PROGRAM P_AxisControl
VAR
END_VAR

//Axis Control program based on youtube series Twincat 3 NC Videos MB05a until MB17b plus MB22 by @electricalautomation https://www.youtube.com/watch?v=BxRAOdTks9I&list=PL762SfoJC-e8NbAUQ-H7a_TOdqrlBPCw4&index=25

IF G_Inputs.bManualModeSelector THEN
	Manual_mode();
ELSIF G_Inputs.bAutoModeSelector THEN
	Auto_mode();
ELSE
	Stop_mode();
END_IF

METHOD Auto_mode : BOOL
VAR_INPUT
END_VAR
//AXIS 1 Main arm actuator

G_AXIS1.lrBC_PowerOverride := 100;

G_AXIS1.bBC_ResetExe := G_Inputs.bJoystickLeftEnable OR G_Inputs.bGreenButton OR G_AXIS1.bBC_MoveAbsDone;

//Power Enable
G_AXIS1.bBC_PowerEnCmd := G_Inputs.bAutoModeSelector;
G_AXIS1.bBC_PowerEnNegative := G_Inputs.bAutoModeSelector;
G_AXIS1.bBC_PowerEnPositive := G_Inputs.bAutoModeSelector;

G_AXIS1.lrBC_MoveAbsPosition := G_InverseKinematics.fStrokeActuatorMainInverse*1000;
G_AXIS1.lrBC_MoveAbsVelocity := 20;
G_AXIS1.bBC_MoveAbsExe := G_Inputs.bGreenButton;


//Position control
IF G_Inputs.bJoystickLeftEnable AND G_AXIS1.bBC_MoveAbsDone THEN
	G_AXIS1.bBC_ExtSetGenDisExe := FALSE;
	G_AXIS1.bBC_ExtSetGenEnaExe := TRUE;
ELSE
	G_AXIS1.bBC_ExtSetGenDisExe := TRUE;
	G_AXIS1.bBC_ExtSetGenEnaExe := FALSE;
END_IF


G_AXIS1.lrBC_MoveAddPos := G_InverseKinematics.fStrokeActuatorMainInverse*1000;


//Update axis
AXIS1_LD_Auto();


//Axis 3 Knuckle arm actuator

G_AXIS3.lrTC_PowerOverride := 100;

G_AXIS3.bTC_ResetExe := G_Inputs.bJoystickLeftEnable OR G_Inputs.bGreenButton OR G_AXIS3.bTC_MoveAbsDone;

//Power Enable
G_AXIS3.bTC_PowerEnCmd := G_Inputs.bAutoModeSelector;
G_AXIS3.bTC_PowerEnNegative := G_Inputs.bAutoModeSelector;
G_AXIS3.bTC_PowerEnPositive := G_Inputs.bAutoModeSelector;

G_AXIS3.lrTC_MoveAbsPosition := G_InverseKinematics.fStrokeActuatorKnuckleInverse*1000;
G_AXIS3.lrTC_MoveAbsVelocity := 20;
G_AXIS3.bTC_MoveAbsExe := G_Inputs.bGreenButton;


//Position control
IF G_Inputs.bJoystickLeftEnable AND G_AXIS3.bTC_MoveAbsDone THEN
	G_AXIS3.bTC_ExtSetGenDisExe := FALSE;
	G_AXIS3.bTC_ExtSetGenEnaExe := TRUE;
ELSE
	G_AXIS3.bTC_ExtSetGenDisExe := TRUE;
	G_AXIS3.bTC_ExtSetGenEnaExe := FALSE;
END_IF


G_AXIS3.lrTC_MoveAddPos := G_InverseKinematics.fStrokeActuatorKnuckleInverse*1000;


//Update axis
AXIS3_LD_Auto();


//Axis 4 Winch motor

G_AXIS4.lrWM_PowerOverride := 50;

G_AXIS4.bWM_ResetExe := G_Inputs.bGreenButton OR G_AXIS1.bBC_MoveAbsDone;
//GVL_AXIS4.bWM_ResetExe := G_Inputs.bJoystickRightEnable OR G_Inputs.bGreenButton OR GVL_AXIS1.bBC_MoveAbsDone;

//Power Enable
G_AXIS4.bWM_PowerEnCmd := G_Inputs.bAutoModeSelector;
G_AXIS4.bWM_PowerEnNegative := G_Inputs.bAutoModeSelector;
G_AXIS4.bWM_PowerEnPositive := G_Inputs.bAutoModeSelector;

//G_AXIS4.lrWM_MoveAbsPosition := G_MachineControl.fWinchMotorAngleRef*180/PI;
//G_AXIS4.lrWM_MoveAbsVelocity := 50;
//G_AXIS4.bWM_MoveAbsExe := G_Inputs.bGreenButton;

//Position control
IF G_Inputs.bJoystickLeftEnable AND G_AXIS1.bBC_MoveAbsDone AND G_AXIS3.bTC_MoveAbsDone THEN
	G_AXIS4.bWM_ExtSetGenDisExe := FALSE;
	G_AXIS4.bWM_ExtSetGenEnaExe := TRUE;
ELSE
	G_AXIS4.bWM_ExtSetGenDisExe := TRUE;
	G_AXIS4.bWM_ExtSetGenEnaExe := FALSE;
END_IF

G_AXIS4.lrWM_MoveSetPointVel := 500;
G_AXIS4.lrWM_MoveAddPos := G_MachineControl.fWinchMotorAngleAbsRef; //G_MachineControl.fWinchMotorAngleRef*180/PI; //Convert to degrees


//Update axis
AXIS4_LD_Auto();
END_METHOD

METHOD AXIS1_LD_Auto : BOOL
VAR_INPUT
END_VAR
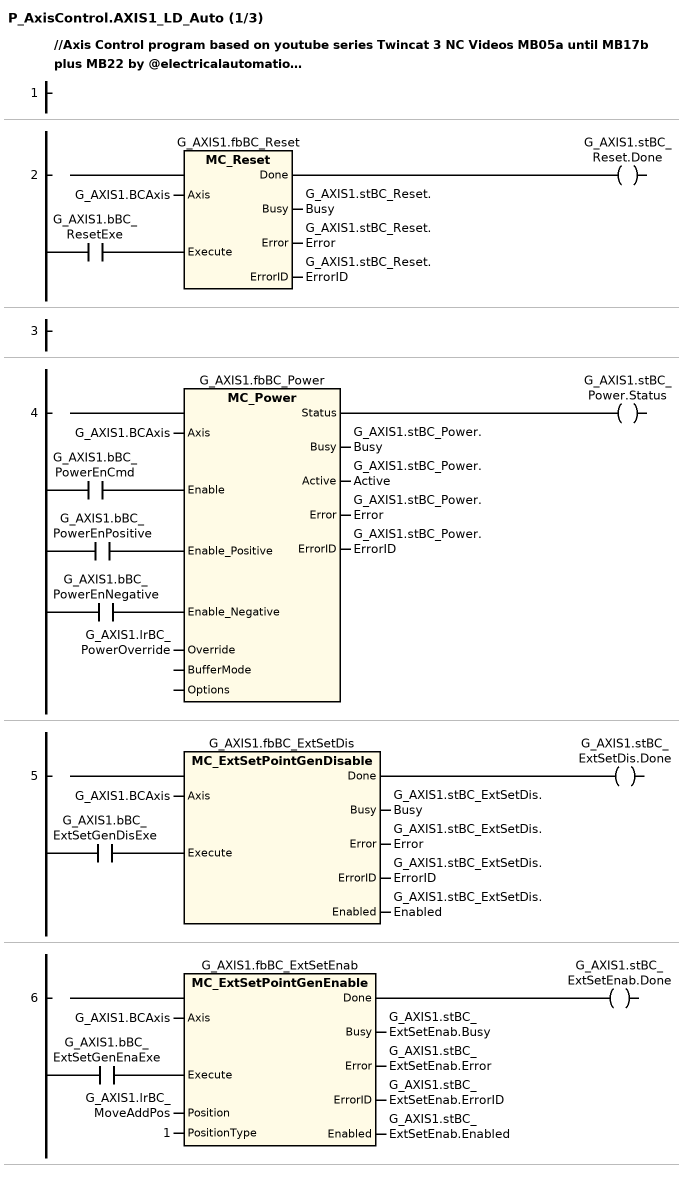
// NETWORK 1: //Axis Control program based on youtube series Twincat 3 NC Videos MB05a until MB17b plus MB22 by @electricalautomation https://www.youtube.com/watch?v=BxRAOdTks9I&list=PL762SfoJC-e8NbAUQ-H7a_TOdqrlBPCw4&index=25

// NETWORK 2
G_AXIS1.fbBC_Reset(
    Axis := G_AXIS1.BCAxis,
    Execute := G_AXIS1.bBC_ResetExe,
    Busy => G_AXIS1.stBC_Reset.Busy,
    Error => G_AXIS1.stBC_Reset.Error,
    ErrorID => G_AXIS1.stBC_Reset.ErrorID); // MC_Reset
G_AXIS1.stBC_Reset.Done := G_AXIS1.fbBC_Reset.Done;

// NETWORK 3

// NETWORK 4
G_AXIS1.fbBC_Power(
    Axis := G_AXIS1.BCAxis,
    Enable := G_AXIS1.bBC_PowerEnCmd,
    Enable_Positive := G_AXIS1.bBC_PowerEnPositive,
    Enable_Negative := G_AXIS1.bBC_PowerEnNegative,
    Override := G_AXIS1.lrBC_PowerOverride,
    Busy => G_AXIS1.stBC_Power.Busy,
    Active => G_AXIS1.stBC_Power.Active,
    Error => G_AXIS1.stBC_Power.Error,
    ErrorID => G_AXIS1.stBC_Power.ErrorID); // MC_Power
G_AXIS1.stBC_Power.Status := G_AXIS1.fbBC_Power.Status;

// NETWORK 5
G_AXIS1.fbBC_ExtSetDis(
    Axis := G_AXIS1.BCAxis,
    Execute := G_AXIS1.bBC_ExtSetGenDisExe,
    Busy => G_AXIS1.stBC_ExtSetDis.Busy,
    Error => G_AXIS1.stBC_ExtSetDis.Error,
    ErrorID => G_AXIS1.stBC_ExtSetDis.ErrorID,
    Enabled => G_AXIS1.stBC_ExtSetDis.Enabled); // MC_ExtSetPointGenDisable
G_AXIS1.stBC_ExtSetDis.Done := G_AXIS1.fbBC_ExtSetDis.Done;

// NETWORK 6
G_AXIS1.fbBC_ExtSetEnab(
    Axis := G_AXIS1.BCAxis,
    Execute := G_AXIS1.bBC_ExtSetGenEnaExe,
    Position := G_AXIS1.lrBC_MoveAddPos,
    PositionType := 1,
    Busy => G_AXIS1.stBC_ExtSetEnab.Busy,
    Error => G_AXIS1.stBC_ExtSetEnab.Error,
    ErrorID => G_AXIS1.stBC_ExtSetEnab.ErrorID,
    Enabled => G_AXIS1.stBC_ExtSetEnab.Enabled); // MC_ExtSetPointGenEnable
G_AXIS1.stBC_ExtSetEnab.Done := G_AXIS1.fbBC_ExtSetEnab.Done;

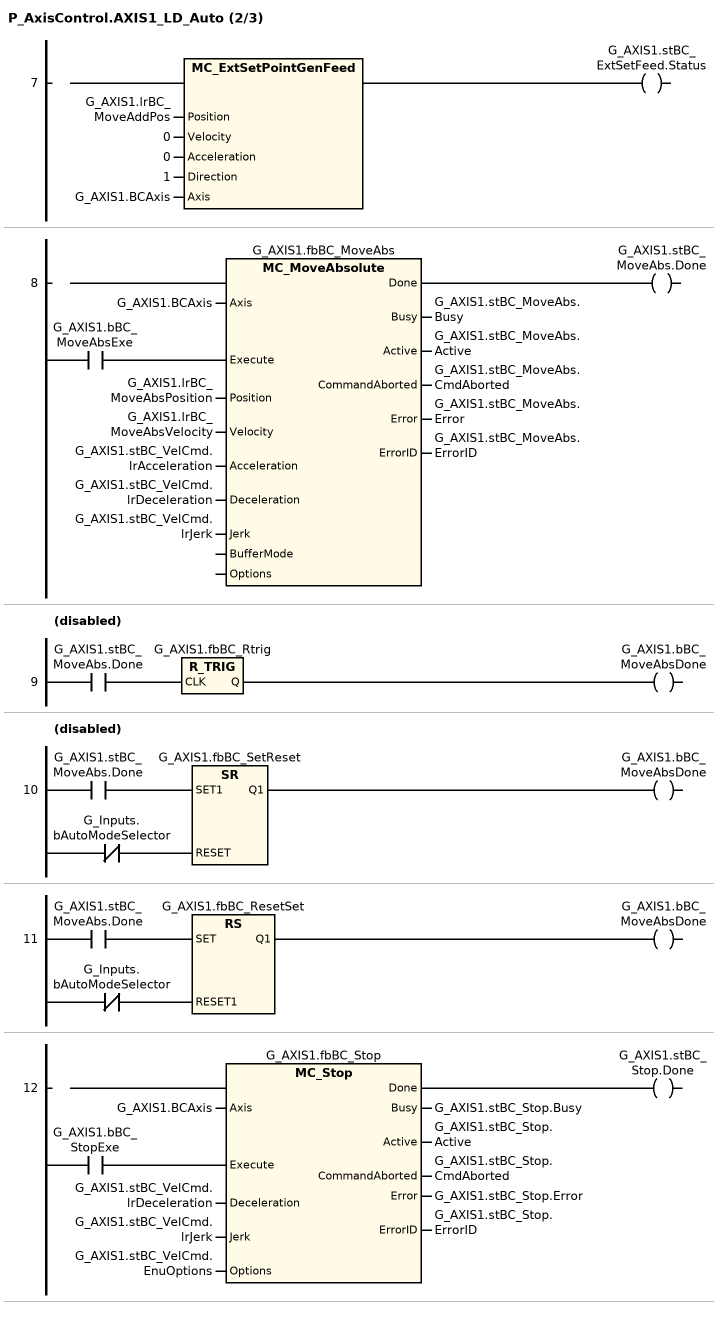
// NETWORK 7
G_AXIS1.stBC_ExtSetFeed.Status := MC_ExtSetPointGenFeed(Position := G_AXIS1.lrBC_MoveAddPos, Velocity := 0, Acceleration := 0, Direction := 1, Axis := G_AXIS1.BCAxis);

// NETWORK 8
G_AXIS1.fbBC_MoveAbs(
    Axis := G_AXIS1.BCAxis,
    Execute := G_AXIS1.bBC_MoveAbsExe,
    Position := G_AXIS1.lrBC_MoveAbsPosition,
    Velocity := G_AXIS1.lrBC_MoveAbsVelocity,
    Acceleration := G_AXIS1.stBC_VelCmd.lrAcceleration,
    Deceleration := G_AXIS1.stBC_VelCmd.lrDeceleration,
    Jerk := G_AXIS1.stBC_VelCmd.lrJerk,
    Busy => G_AXIS1.stBC_MoveAbs.Busy,
    Active => G_AXIS1.stBC_MoveAbs.Active,
    CommandAborted => G_AXIS1.stBC_MoveAbs.CmdAborted,
    Error => G_AXIS1.stBC_MoveAbs.Error,
    ErrorID => G_AXIS1.stBC_MoveAbs.ErrorID); // MC_MoveAbsolute
G_AXIS1.stBC_MoveAbs.Done := G_AXIS1.fbBC_MoveAbs.Done;

// NETWORK 9 (disabled)
// G_AXIS1.fbBC_Rtrig(CLK := G_AXIS1.stBC_MoveAbs.Done); // R_TRIG
// G_AXIS1.bBC_MoveAbsDone := G_AXIS1.fbBC_Rtrig.Q;

// NETWORK 10 (disabled)
// G_AXIS1.fbBC_SetReset(SET1 := G_AXIS1.stBC_MoveAbs.Done, RESET := NOT G_Inputs.bAutoModeSelector); // SR
// G_AXIS1.bBC_MoveAbsDone := G_AXIS1.fbBC_SetReset.Q1;

// NETWORK 11
G_AXIS1.fbBC_ResetSet(SET := G_AXIS1.stBC_MoveAbs.Done, RESET1 := NOT G_Inputs.bAutoModeSelector); // RS
G_AXIS1.bBC_MoveAbsDone := G_AXIS1.fbBC_ResetSet.Q1;

// NETWORK 12
G_AXIS1.fbBC_Stop(
    Axis := G_AXIS1.BCAxis,
    Execute := G_AXIS1.bBC_StopExe,
    Deceleration := G_AXIS1.stBC_VelCmd.lrDeceleration,
    Jerk := G_AXIS1.stBC_VelCmd.lrJerk,
    Options := G_AXIS1.stBC_VelCmd.EnuOptions,
    Busy => G_AXIS1.stBC_Stop.Busy,
    Active => G_AXIS1.stBC_Stop.Active,
    CommandAborted => G_AXIS1.stBC_Stop.CmdAborted,
    Error => G_AXIS1.stBC_Stop.Error,
    ErrorID => G_AXIS1.stBC_Stop.ErrorID); // MC_Stop
G_AXIS1.stBC_Stop.Done := G_AXIS1.fbBC_Stop.Done;

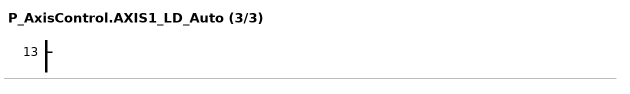
// NETWORK 13
END_METHOD

METHOD AXIS1_LD_Manual : BOOL
VAR_INPUT
END_VAR
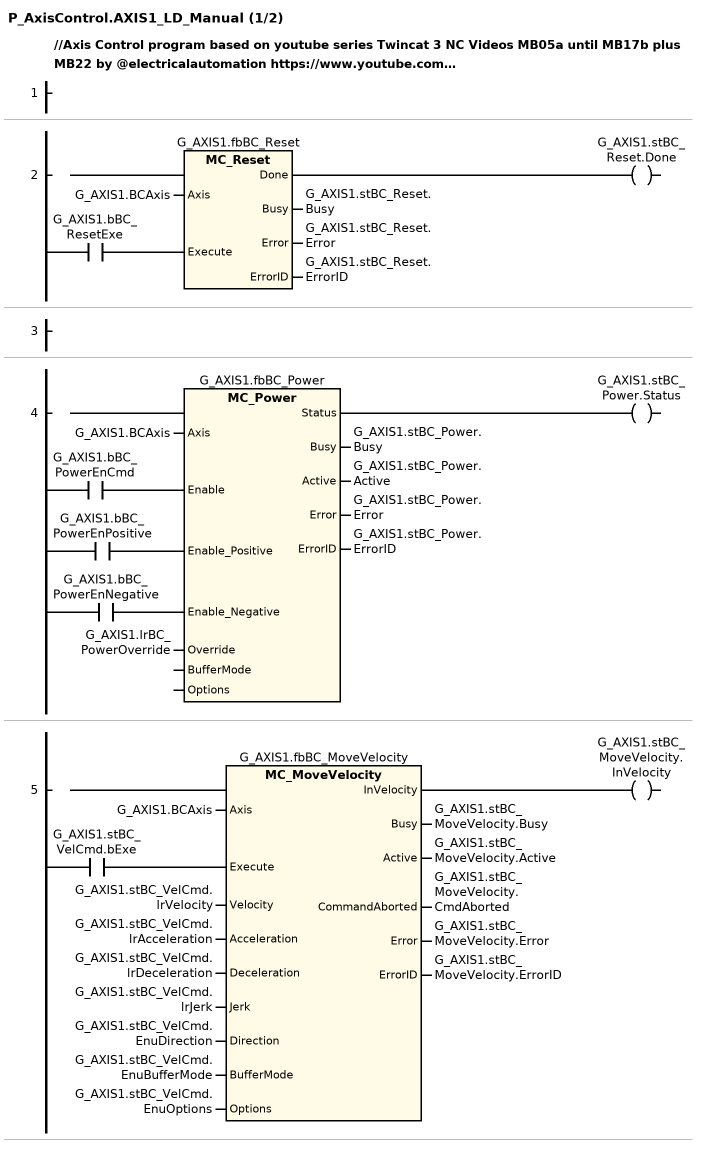
// NETWORK 1: //Axis Control program based on youtube series Twincat 3 NC Videos MB05a until MB17b plus MB22 by @electricalautomation https://www.youtube.com/watch?v=BxRAOdTks9I&list=PL762SfoJC-e8NbAUQ-H7a_TOdqrlBPCw4&index=25

// NETWORK 2
G_AXIS1.fbBC_Reset(
    Axis := G_AXIS1.BCAxis,
    Execute := G_AXIS1.bBC_ResetExe,
    Busy => G_AXIS1.stBC_Reset.Busy,
    Error => G_AXIS1.stBC_Reset.Error,
    ErrorID => G_AXIS1.stBC_Reset.ErrorID); // MC_Reset
G_AXIS1.stBC_Reset.Done := G_AXIS1.fbBC_Reset.Done;

// NETWORK 3

// NETWORK 4
G_AXIS1.fbBC_Power(
    Axis := G_AXIS1.BCAxis,
    Enable := G_AXIS1.bBC_PowerEnCmd,
    Enable_Positive := G_AXIS1.bBC_PowerEnPositive,
    Enable_Negative := G_AXIS1.bBC_PowerEnNegative,
    Override := G_AXIS1.lrBC_PowerOverride,
    Busy => G_AXIS1.stBC_Power.Busy,
    Active => G_AXIS1.stBC_Power.Active,
    Error => G_AXIS1.stBC_Power.Error,
    ErrorID => G_AXIS1.stBC_Power.ErrorID); // MC_Power
G_AXIS1.stBC_Power.Status := G_AXIS1.fbBC_Power.Status;

// NETWORK 5
G_AXIS1.fbBC_MoveVelocity(
    Axis := G_AXIS1.BCAxis,
    Execute := G_AXIS1.stBC_VelCmd.bExe,
    Velocity := G_AXIS1.stBC_VelCmd.lrVelocity,
    Acceleration := G_AXIS1.stBC_VelCmd.lrAcceleration,
    Deceleration := G_AXIS1.stBC_VelCmd.lrDeceleration,
    Jerk := G_AXIS1.stBC_VelCmd.lrJerk,
    Direction := G_AXIS1.stBC_VelCmd.EnuDirection,
    BufferMode := G_AXIS1.stBC_VelCmd.EnuBufferMode,
    Options := G_AXIS1.stBC_VelCmd.EnuOptions,
    Busy => G_AXIS1.stBC_MoveVelocity.Busy,
    Active => G_AXIS1.stBC_MoveVelocity.Active,
    CommandAborted => G_AXIS1.stBC_MoveVelocity.CmdAborted,
    Error => G_AXIS1.stBC_MoveVelocity.Error,
    ErrorID => G_AXIS1.stBC_MoveVelocity.ErrorID); // MC_MoveVelocity
G_AXIS1.stBC_MoveVelocity.InVelocity := G_AXIS1.fbBC_MoveVelocity.InVelocity;

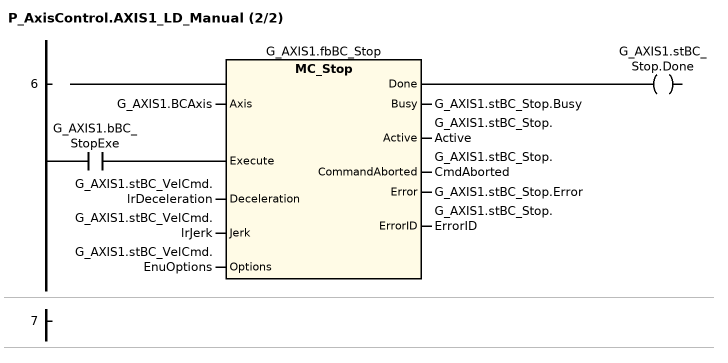
// NETWORK 6
G_AXIS1.fbBC_Stop(
    Axis := G_AXIS1.BCAxis,
    Execute := G_AXIS1.bBC_StopExe,
    Deceleration := G_AXIS1.stBC_VelCmd.lrDeceleration,
    Jerk := G_AXIS1.stBC_VelCmd.lrJerk,
    Options := G_AXIS1.stBC_VelCmd.EnuOptions,
    Busy => G_AXIS1.stBC_Stop.Busy,
    Active => G_AXIS1.stBC_Stop.Active,
    CommandAborted => G_AXIS1.stBC_Stop.CmdAborted,
    Error => G_AXIS1.stBC_Stop.Error,
    ErrorID => G_AXIS1.stBC_Stop.ErrorID); // MC_Stop
G_AXIS1.stBC_Stop.Done := G_AXIS1.fbBC_Stop.Done;

// NETWORK 7
END_METHOD

METHOD AXIS2_LD_Manual : BOOL
VAR_INPUT
END_VAR
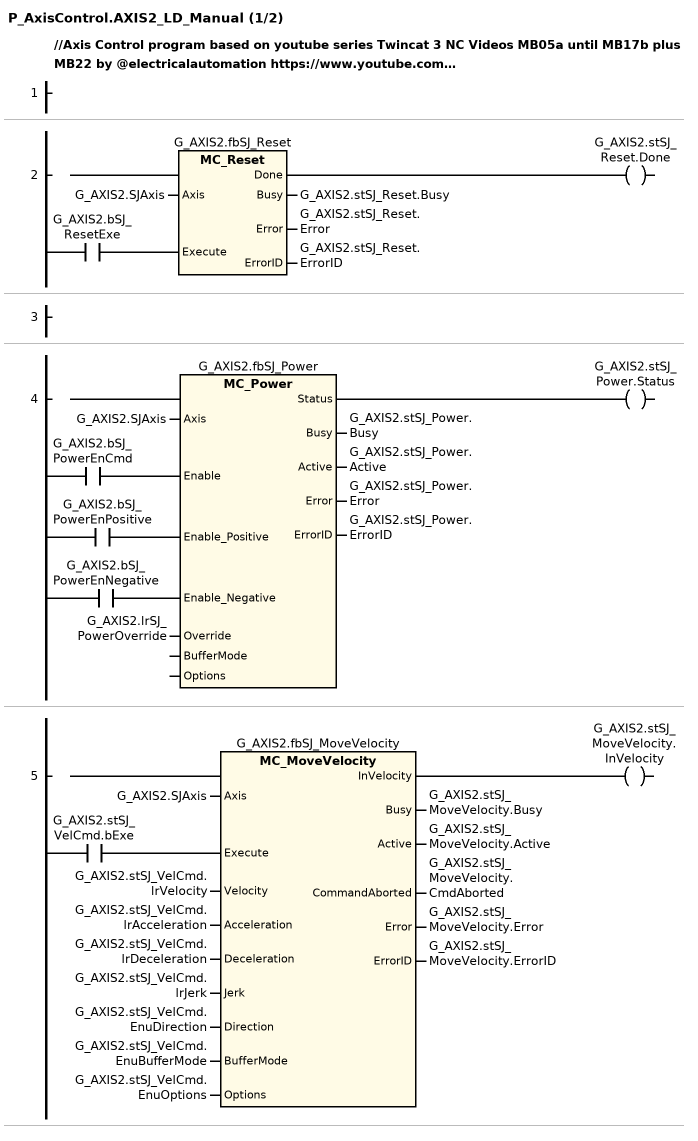
// NETWORK 1: //Axis Control program based on youtube series Twincat 3 NC Videos MB05a until MB17b plus MB22 by @electricalautomation https://www.youtube.com/watch?v=BxRAOdTks9I&list=PL762SfoJC-e8NbAUQ-H7a_TOdqrlBPCw4&index=25

// NETWORK 2
G_AXIS2.fbSJ_Reset(
    Axis := G_AXIS2.SJAxis,
    Execute := G_AXIS2.bSJ_ResetExe,
    Busy => G_AXIS2.stSJ_Reset.Busy,
    Error => G_AXIS2.stSJ_Reset.Error,
    ErrorID => G_AXIS2.stSJ_Reset.ErrorID); // MC_Reset
G_AXIS2.stSJ_Reset.Done := G_AXIS2.fbSJ_Reset.Done;

// NETWORK 3

// NETWORK 4
G_AXIS2.fbSJ_Power(
    Axis := G_AXIS2.SJAxis,
    Enable := G_AXIS2.bSJ_PowerEnCmd,
    Enable_Positive := G_AXIS2.bSJ_PowerEnPositive,
    Enable_Negative := G_AXIS2.bSJ_PowerEnNegative,
    Override := G_AXIS2.lrSJ_PowerOverride,
    Busy => G_AXIS2.stSJ_Power.Busy,
    Active => G_AXIS2.stSJ_Power.Active,
    Error => G_AXIS2.stSJ_Power.Error,
    ErrorID => G_AXIS2.stSJ_Power.ErrorID); // MC_Power
G_AXIS2.stSJ_Power.Status := G_AXIS2.fbSJ_Power.Status;

// NETWORK 5
G_AXIS2.fbSJ_MoveVelocity(
    Axis := G_AXIS2.SJAxis,
    Execute := G_AXIS2.stSJ_VelCmd.bExe,
    Velocity := G_AXIS2.stSJ_VelCmd.lrVelocity,
    Acceleration := G_AXIS2.stSJ_VelCmd.lrAcceleration,
    Deceleration := G_AXIS2.stSJ_VelCmd.lrDeceleration,
    Jerk := G_AXIS2.stSJ_VelCmd.lrJerk,
    Direction := G_AXIS2.stSJ_VelCmd.EnuDirection,
    BufferMode := G_AXIS2.stSJ_VelCmd.EnuBufferMode,
    Options := G_AXIS2.stSJ_VelCmd.EnuOptions,
    Busy => G_AXIS2.stSJ_MoveVelocity.Busy,
    Active => G_AXIS2.stSJ_MoveVelocity.Active,
    CommandAborted => G_AXIS2.stSJ_MoveVelocity.CmdAborted,
    Error => G_AXIS2.stSJ_MoveVelocity.Error,
    ErrorID => G_AXIS2.stSJ_MoveVelocity.ErrorID); // MC_MoveVelocity
G_AXIS2.stSJ_MoveVelocity.InVelocity := G_AXIS2.fbSJ_MoveVelocity.InVelocity;

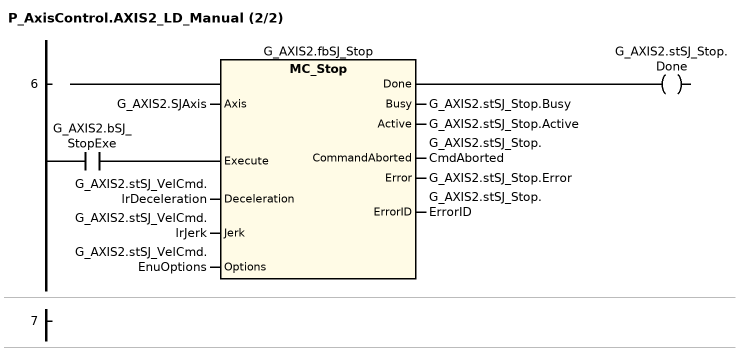
// NETWORK 6
G_AXIS2.fbSJ_Stop(
    Axis := G_AXIS2.SJAxis,
    Execute := G_AXIS2.bSJ_StopExe,
    Deceleration := G_AXIS2.stSJ_VelCmd.lrDeceleration,
    Jerk := G_AXIS2.stSJ_VelCmd.lrJerk,
    Options := G_AXIS2.stSJ_VelCmd.EnuOptions,
    Busy => G_AXIS2.stSJ_Stop.Busy,
    Active => G_AXIS2.stSJ_Stop.Active,
    CommandAborted => G_AXIS2.stSJ_Stop.CmdAborted,
    Error => G_AXIS2.stSJ_Stop.Error,
    ErrorID => G_AXIS2.stSJ_Stop.ErrorID); // MC_Stop
G_AXIS2.stSJ_Stop.Done := G_AXIS2.fbSJ_Stop.Done;

// NETWORK 7
END_METHOD

METHOD AXIS3_LD_Auto : BOOL
VAR_INPUT
END_VAR
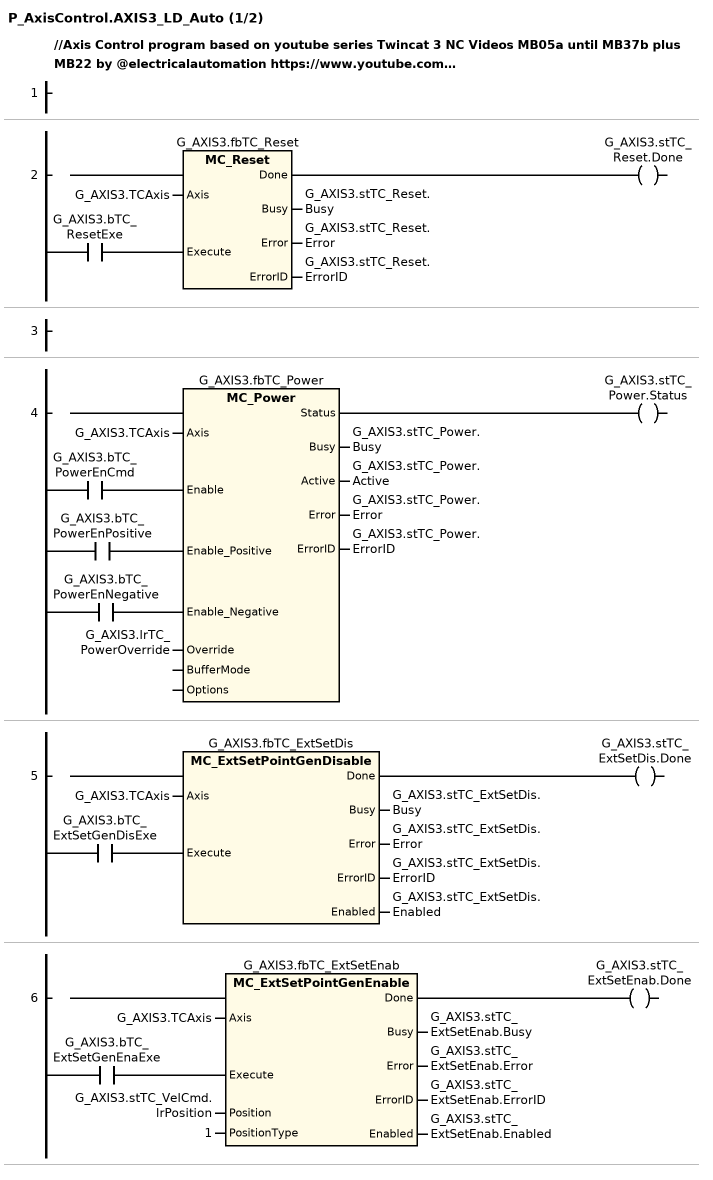
// NETWORK 1: //Axis Control program based on youtube series Twincat 3 NC Videos MB05a until MB37b plus MB22 by @electricalautomation https://www.youtube.com/watch?v=BxRAOdTks9I&list=PL762SfoJC-e8NbAUQ-H7a_TOdqrlBPCw4&index=25

// NETWORK 2
G_AXIS3.fbTC_Reset(
    Axis := G_AXIS3.TCAxis,
    Execute := G_AXIS3.bTC_ResetExe,
    Busy => G_AXIS3.stTC_Reset.Busy,
    Error => G_AXIS3.stTC_Reset.Error,
    ErrorID => G_AXIS3.stTC_Reset.ErrorID); // MC_Reset
G_AXIS3.stTC_Reset.Done := G_AXIS3.fbTC_Reset.Done;

// NETWORK 3

// NETWORK 4
G_AXIS3.fbTC_Power(
    Axis := G_AXIS3.TCAxis,
    Enable := G_AXIS3.bTC_PowerEnCmd,
    Enable_Positive := G_AXIS3.bTC_PowerEnPositive,
    Enable_Negative := G_AXIS3.bTC_PowerEnNegative,
    Override := G_AXIS3.lrTC_PowerOverride,
    Busy => G_AXIS3.stTC_Power.Busy,
    Active => G_AXIS3.stTC_Power.Active,
    Error => G_AXIS3.stTC_Power.Error,
    ErrorID => G_AXIS3.stTC_Power.ErrorID); // MC_Power
G_AXIS3.stTC_Power.Status := G_AXIS3.fbTC_Power.Status;

// NETWORK 5
G_AXIS3.fbTC_ExtSetDis(
    Axis := G_AXIS3.TCAxis,
    Execute := G_AXIS3.bTC_ExtSetGenDisExe,
    Busy => G_AXIS3.stTC_ExtSetDis.Busy,
    Error => G_AXIS3.stTC_ExtSetDis.Error,
    ErrorID => G_AXIS3.stTC_ExtSetDis.ErrorID,
    Enabled => G_AXIS3.stTC_ExtSetDis.Enabled); // MC_ExtSetPointGenDisable
G_AXIS3.stTC_ExtSetDis.Done := G_AXIS3.fbTC_ExtSetDis.Done;

// NETWORK 6
G_AXIS3.fbTC_ExtSetEnab(
    Axis := G_AXIS3.TCAxis,
    Execute := G_AXIS3.bTC_ExtSetGenEnaExe,
    Position := G_AXIS3.stTC_VelCmd.lrPosition,
    PositionType := 1,
    Busy => G_AXIS3.stTC_ExtSetEnab.Busy,
    Error => G_AXIS3.stTC_ExtSetEnab.Error,
    ErrorID => G_AXIS3.stTC_ExtSetEnab.ErrorID,
    Enabled => G_AXIS3.stTC_ExtSetEnab.Enabled); // MC_ExtSetPointGenEnable
G_AXIS3.stTC_ExtSetEnab.Done := G_AXIS3.fbTC_ExtSetEnab.Done;

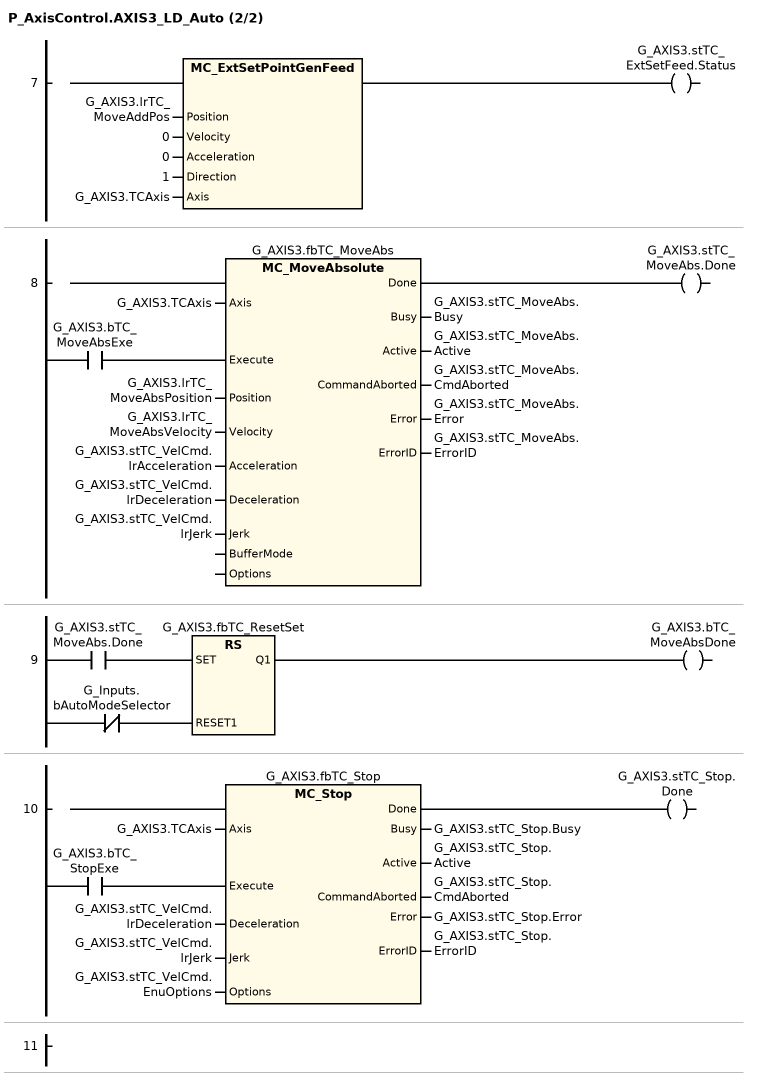
// NETWORK 7
G_AXIS3.stTC_ExtSetFeed.Status := MC_ExtSetPointGenFeed(Position := G_AXIS3.lrTC_MoveAddPos, Velocity := 0, Acceleration := 0, Direction := 1, Axis := G_AXIS3.TCAxis);

// NETWORK 8
G_AXIS3.fbTC_MoveAbs(
    Axis := G_AXIS3.TCAxis,
    Execute := G_AXIS3.bTC_MoveAbsExe,
    Position := G_AXIS3.lrTC_MoveAbsPosition,
    Velocity := G_AXIS3.lrTC_MoveAbsVelocity,
    Acceleration := G_AXIS3.stTC_VelCmd.lrAcceleration,
    Deceleration := G_AXIS3.stTC_VelCmd.lrDeceleration,
    Jerk := G_AXIS3.stTC_VelCmd.lrJerk,
    Busy => G_AXIS3.stTC_MoveAbs.Busy,
    Active => G_AXIS3.stTC_MoveAbs.Active,
    CommandAborted => G_AXIS3.stTC_MoveAbs.CmdAborted,
    Error => G_AXIS3.stTC_MoveAbs.Error,
    ErrorID => G_AXIS3.stTC_MoveAbs.ErrorID); // MC_MoveAbsolute
G_AXIS3.stTC_MoveAbs.Done := G_AXIS3.fbTC_MoveAbs.Done;

// NETWORK 9
G_AXIS3.fbTC_ResetSet(SET := G_AXIS3.stTC_MoveAbs.Done, RESET1 := NOT G_Inputs.bAutoModeSelector); // RS
G_AXIS3.bTC_MoveAbsDone := G_AXIS3.fbTC_ResetSet.Q1;

// NETWORK 10
G_AXIS3.fbTC_Stop(
    Axis := G_AXIS3.TCAxis,
    Execute := G_AXIS3.bTC_StopExe,
    Deceleration := G_AXIS3.stTC_VelCmd.lrDeceleration,
    Jerk := G_AXIS3.stTC_VelCmd.lrJerk,
    Options := G_AXIS3.stTC_VelCmd.EnuOptions,
    Busy => G_AXIS3.stTC_Stop.Busy,
    Active => G_AXIS3.stTC_Stop.Active,
    CommandAborted => G_AXIS3.stTC_Stop.CmdAborted,
    Error => G_AXIS3.stTC_Stop.Error,
    ErrorID => G_AXIS3.stTC_Stop.ErrorID); // MC_Stop
G_AXIS3.stTC_Stop.Done := G_AXIS3.fbTC_Stop.Done;

// NETWORK 11
END_METHOD

METHOD AXIS3_LD_Manual : BOOL
VAR_INPUT
END_VAR
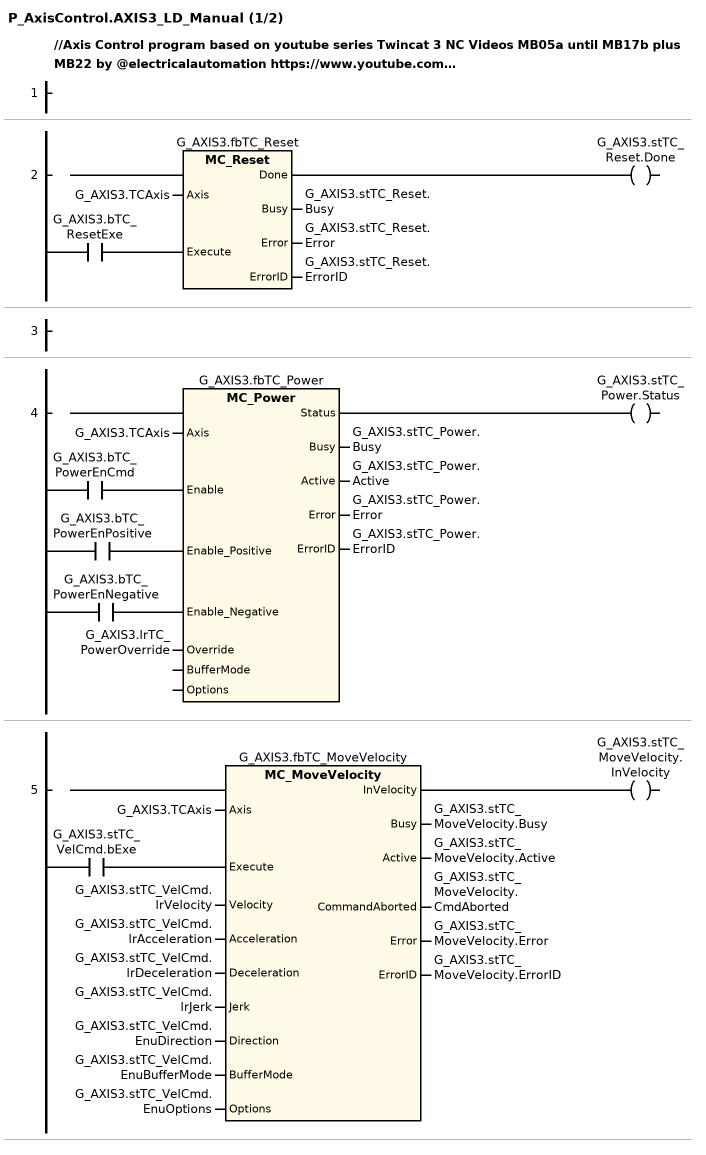
// NETWORK 1: //Axis Control program based on youtube series Twincat 3 NC Videos MB05a until MB17b plus MB22 by @electricalautomation https://www.youtube.com/watch?v=BxRAOdTks9I&list=PL762SfoJC-e8NbAUQ-H7a_TOdqrlBPCw4&index=25

// NETWORK 2
G_AXIS3.fbTC_Reset(
    Axis := G_AXIS3.TCAxis,
    Execute := G_AXIS3.bTC_ResetExe,
    Busy => G_AXIS3.stTC_Reset.Busy,
    Error => G_AXIS3.stTC_Reset.Error,
    ErrorID => G_AXIS3.stTC_Reset.ErrorID); // MC_Reset
G_AXIS3.stTC_Reset.Done := G_AXIS3.fbTC_Reset.Done;

// NETWORK 3

// NETWORK 4
G_AXIS3.fbTC_Power(
    Axis := G_AXIS3.TCAxis,
    Enable := G_AXIS3.bTC_PowerEnCmd,
    Enable_Positive := G_AXIS3.bTC_PowerEnPositive,
    Enable_Negative := G_AXIS3.bTC_PowerEnNegative,
    Override := G_AXIS3.lrTC_PowerOverride,
    Busy => G_AXIS3.stTC_Power.Busy,
    Active => G_AXIS3.stTC_Power.Active,
    Error => G_AXIS3.stTC_Power.Error,
    ErrorID => G_AXIS3.stTC_Power.ErrorID); // MC_Power
G_AXIS3.stTC_Power.Status := G_AXIS3.fbTC_Power.Status;

// NETWORK 5
G_AXIS3.fbTC_MoveVelocity(
    Axis := G_AXIS3.TCAxis,
    Execute := G_AXIS3.stTC_VelCmd.bExe,
    Velocity := G_AXIS3.stTC_VelCmd.lrVelocity,
    Acceleration := G_AXIS3.stTC_VelCmd.lrAcceleration,
    Deceleration := G_AXIS3.stTC_VelCmd.lrDeceleration,
    Jerk := G_AXIS3.stTC_VelCmd.lrJerk,
    Direction := G_AXIS3.stTC_VelCmd.EnuDirection,
    BufferMode := G_AXIS3.stTC_VelCmd.EnuBufferMode,
    Options := G_AXIS3.stTC_VelCmd.EnuOptions,
    Busy => G_AXIS3.stTC_MoveVelocity.Busy,
    Active => G_AXIS3.stTC_MoveVelocity.Active,
    CommandAborted => G_AXIS3.stTC_MoveVelocity.CmdAborted,
    Error => G_AXIS3.stTC_MoveVelocity.Error,
    ErrorID => G_AXIS3.stTC_MoveVelocity.ErrorID); // MC_MoveVelocity
G_AXIS3.stTC_MoveVelocity.InVelocity := G_AXIS3.fbTC_MoveVelocity.InVelocity;

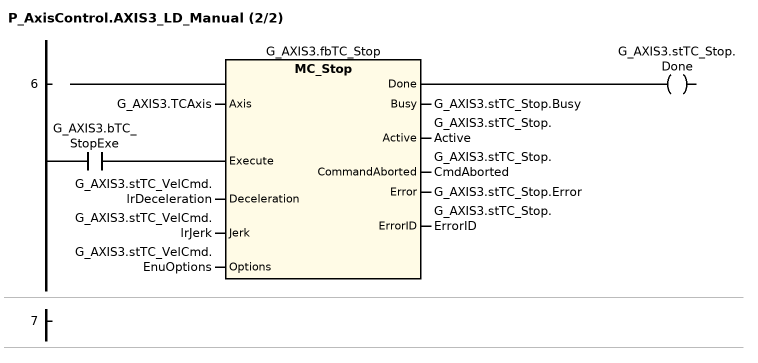
// NETWORK 6
G_AXIS3.fbTC_Stop(
    Axis := G_AXIS3.TCAxis,
    Execute := G_AXIS3.bTC_StopExe,
    Deceleration := G_AXIS3.stTC_VelCmd.lrDeceleration,
    Jerk := G_AXIS3.stTC_VelCmd.lrJerk,
    Options := G_AXIS3.stTC_VelCmd.EnuOptions,
    Busy => G_AXIS3.stTC_Stop.Busy,
    Active => G_AXIS3.stTC_Stop.Active,
    CommandAborted => G_AXIS3.stTC_Stop.CmdAborted,
    Error => G_AXIS3.stTC_Stop.Error,
    ErrorID => G_AXIS3.stTC_Stop.ErrorID); // MC_Stop
G_AXIS3.stTC_Stop.Done := G_AXIS3.fbTC_Stop.Done;

// NETWORK 7
END_METHOD

METHOD AXIS4_LD_Auto : BOOL
VAR_INPUT
END_VAR
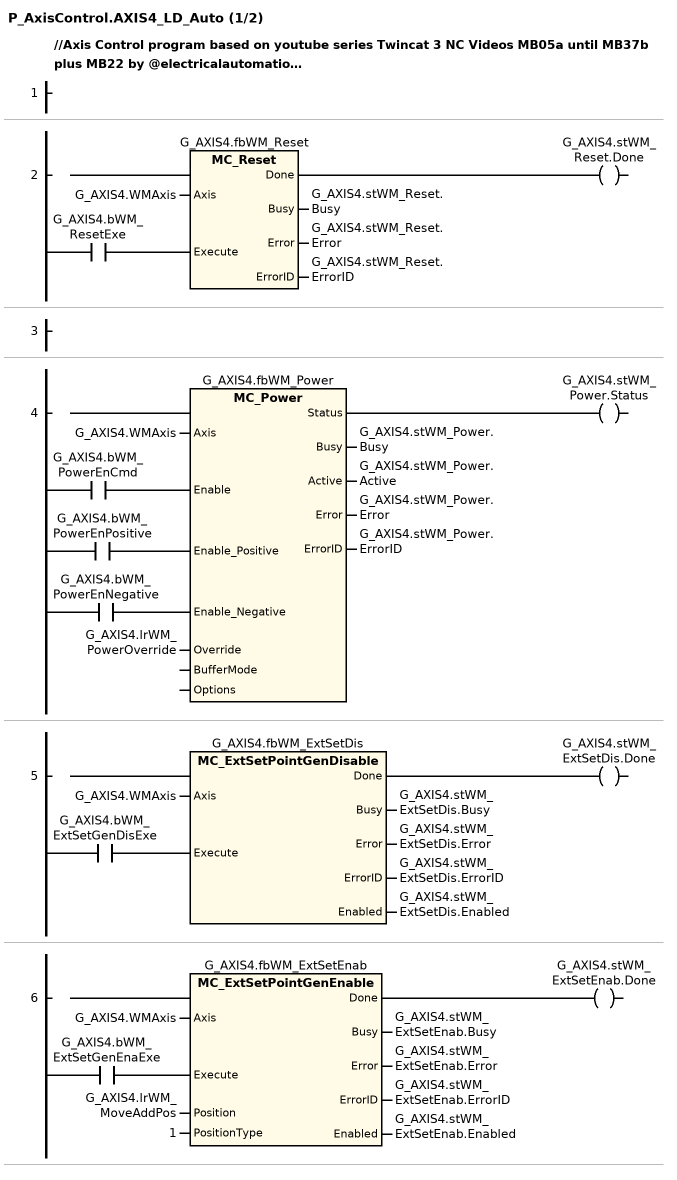
// NETWORK 1: //Axis Control program based on youtube series Twincat 3 NC Videos MB05a until MB37b plus MB22 by @electricalautomation https://www.youtube.com/waWMh?v=BxRAOdTks9I&list=PL762SfoJC-e8NbAUQ-H7a_TOdqrlBPCw4&index=25

// NETWORK 2
G_AXIS4.fbWM_Reset(
    Axis := G_AXIS4.WMAxis,
    Execute := G_AXIS4.bWM_ResetExe,
    Busy => G_AXIS4.stWM_Reset.Busy,
    Error => G_AXIS4.stWM_Reset.Error,
    ErrorID => G_AXIS4.stWM_Reset.ErrorID); // MC_Reset
G_AXIS4.stWM_Reset.Done := G_AXIS4.fbWM_Reset.Done;

// NETWORK 3

// NETWORK 4
G_AXIS4.fbWM_Power(
    Axis := G_AXIS4.WMAxis,
    Enable := G_AXIS4.bWM_PowerEnCmd,
    Enable_Positive := G_AXIS4.bWM_PowerEnPositive,
    Enable_Negative := G_AXIS4.bWM_PowerEnNegative,
    Override := G_AXIS4.lrWM_PowerOverride,
    Busy => G_AXIS4.stWM_Power.Busy,
    Active => G_AXIS4.stWM_Power.Active,
    Error => G_AXIS4.stWM_Power.Error,
    ErrorID => G_AXIS4.stWM_Power.ErrorID); // MC_Power
G_AXIS4.stWM_Power.Status := G_AXIS4.fbWM_Power.Status;

// NETWORK 5
G_AXIS4.fbWM_ExtSetDis(
    Axis := G_AXIS4.WMAxis,
    Execute := G_AXIS4.bWM_ExtSetGenDisExe,
    Busy => G_AXIS4.stWM_ExtSetDis.Busy,
    Error => G_AXIS4.stWM_ExtSetDis.Error,
    ErrorID => G_AXIS4.stWM_ExtSetDis.ErrorID,
    Enabled => G_AXIS4.stWM_ExtSetDis.Enabled); // MC_ExtSetPointGenDisable
G_AXIS4.stWM_ExtSetDis.Done := G_AXIS4.fbWM_ExtSetDis.Done;

// NETWORK 6
G_AXIS4.fbWM_ExtSetEnab(
    Axis := G_AXIS4.WMAxis,
    Execute := G_AXIS4.bWM_ExtSetGenEnaExe,
    Position := G_AXIS4.lrWM_MoveAddPos,
    PositionType := 1,
    Busy => G_AXIS4.stWM_ExtSetEnab.Busy,
    Error => G_AXIS4.stWM_ExtSetEnab.Error,
    ErrorID => G_AXIS4.stWM_ExtSetEnab.ErrorID,
    Enabled => G_AXIS4.stWM_ExtSetEnab.Enabled); // MC_ExtSetPointGenEnable
G_AXIS4.stWM_ExtSetEnab.Done := G_AXIS4.fbWM_ExtSetEnab.Done;

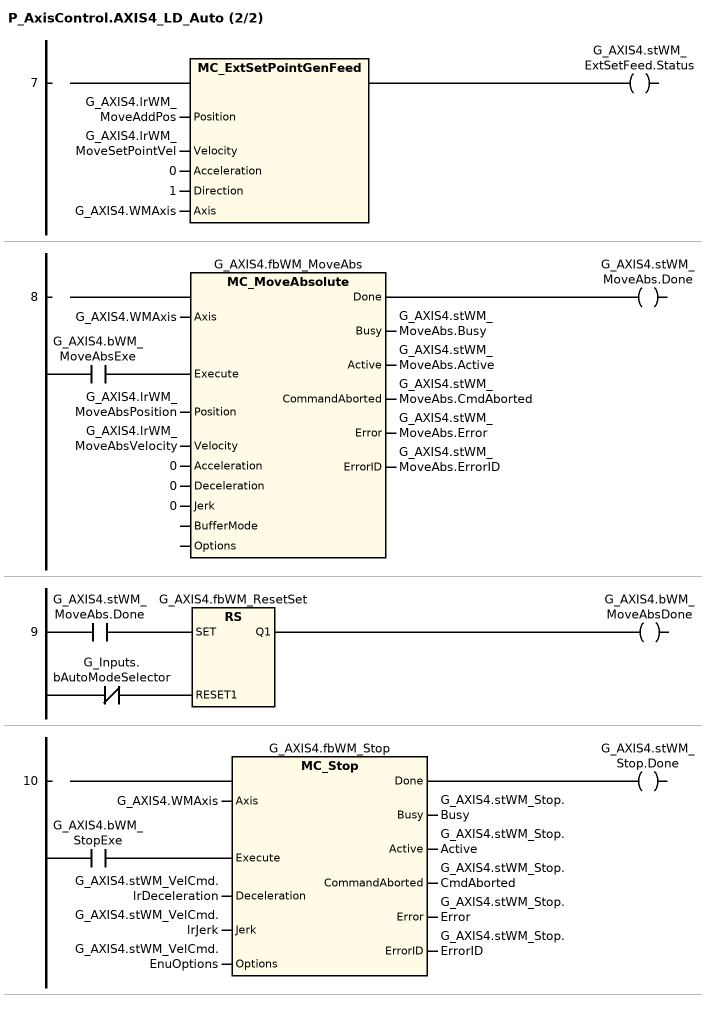
// NETWORK 7
G_AXIS4.stWM_ExtSetFeed.Status := MC_ExtSetPointGenFeed(Position := G_AXIS4.lrWM_MoveAddPos, Velocity := G_AXIS4.lrWM_MoveSetPointVel, Acceleration := 0, Direction := 1, Axis := G_AXIS4.WMAxis);

// NETWORK 8
G_AXIS4.fbWM_MoveAbs(
    Axis := G_AXIS4.WMAxis,
    Execute := G_AXIS4.bWM_MoveAbsExe,
    Position := G_AXIS4.lrWM_MoveAbsPosition,
    Velocity := G_AXIS4.lrWM_MoveAbsVelocity,
    Acceleration := 0,
    Deceleration := 0,
    Jerk := 0,
    Busy => G_AXIS4.stWM_MoveAbs.Busy,
    Active => G_AXIS4.stWM_MoveAbs.Active,
    CommandAborted => G_AXIS4.stWM_MoveAbs.CmdAborted,
    Error => G_AXIS4.stWM_MoveAbs.Error,
    ErrorID => G_AXIS4.stWM_MoveAbs.ErrorID); // MC_MoveAbsolute
G_AXIS4.stWM_MoveAbs.Done := G_AXIS4.fbWM_MoveAbs.Done;

// NETWORK 9
G_AXIS4.fbWM_ResetSet(SET := G_AXIS4.stWM_MoveAbs.Done, RESET1 := NOT G_Inputs.bAutoModeSelector); // RS
G_AXIS4.bWM_MoveAbsDone := G_AXIS4.fbWM_ResetSet.Q1;

// NETWORK 10
G_AXIS4.fbWM_Stop(
    Axis := G_AXIS4.WMAxis,
    Execute := G_AXIS4.bWM_StopExe,
    Deceleration := G_AXIS4.stWM_VelCmd.lrDeceleration,
    Jerk := G_AXIS4.stWM_VelCmd.lrJerk,
    Options := G_AXIS4.stWM_VelCmd.EnuOptions,
    Busy => G_AXIS4.stWM_Stop.Busy,
    Active => G_AXIS4.stWM_Stop.Active,
    CommandAborted => G_AXIS4.stWM_Stop.CmdAborted,
    Error => G_AXIS4.stWM_Stop.Error,
    ErrorID => G_AXIS4.stWM_Stop.ErrorID); // MC_Stop
G_AXIS4.stWM_Stop.Done := G_AXIS4.fbWM_Stop.Done;
END_METHOD

METHOD AXIS4_LD_Manual : BOOL
VAR_INPUT
END_VAR
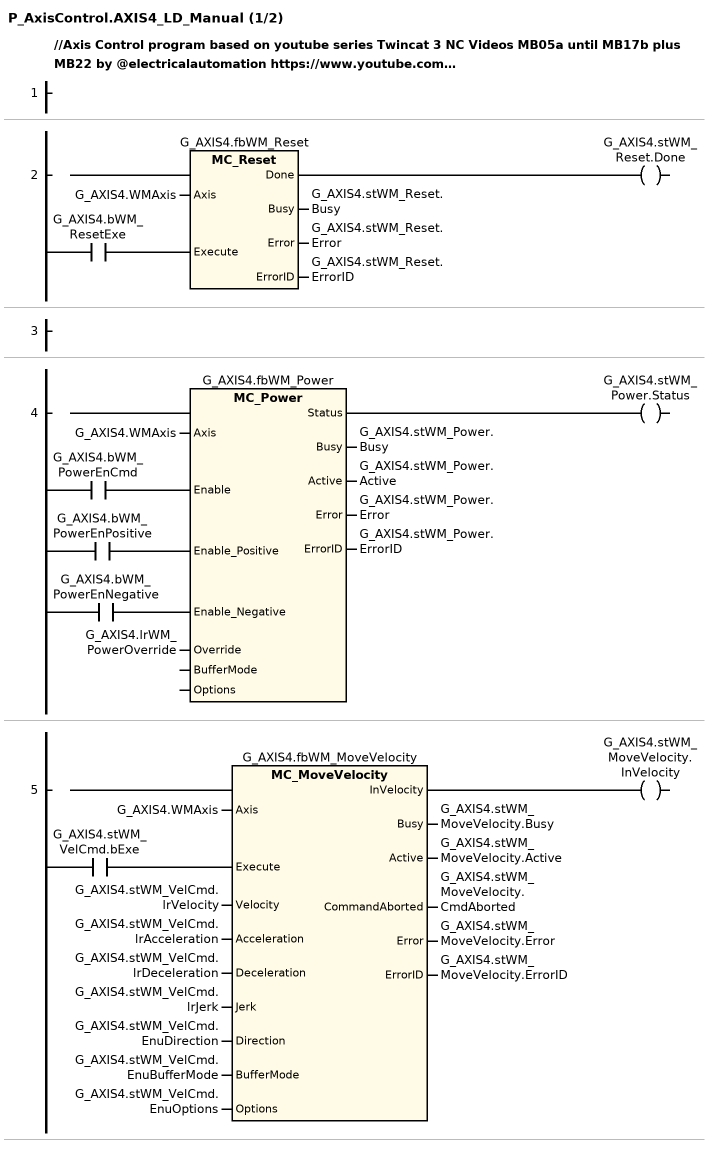
// NETWORK 1: //Axis Control program based on youtube series Twincat 3 NC Videos MB05a until MB17b plus MB22 by @electricalautomation https://www.youtube.com/watch?v=BxRAOdTks9I&list=PL762SfoJC-e8NbAUQ-H7a_TOdqrlBPCw4&index=25

// NETWORK 2
G_AXIS4.fbWM_Reset(
    Axis := G_AXIS4.WMAxis,
    Execute := G_AXIS4.bWM_ResetExe,
    Busy => G_AXIS4.stWM_Reset.Busy,
    Error => G_AXIS4.stWM_Reset.Error,
    ErrorID => G_AXIS4.stWM_Reset.ErrorID); // MC_Reset
G_AXIS4.stWM_Reset.Done := G_AXIS4.fbWM_Reset.Done;

// NETWORK 3

// NETWORK 4
G_AXIS4.fbWM_Power(
    Axis := G_AXIS4.WMAxis,
    Enable := G_AXIS4.bWM_PowerEnCmd,
    Enable_Positive := G_AXIS4.bWM_PowerEnPositive,
    Enable_Negative := G_AXIS4.bWM_PowerEnNegative,
    Override := G_AXIS4.lrWM_PowerOverride,
    Busy => G_AXIS4.stWM_Power.Busy,
    Active => G_AXIS4.stWM_Power.Active,
    Error => G_AXIS4.stWM_Power.Error,
    ErrorID => G_AXIS4.stWM_Power.ErrorID); // MC_Power
G_AXIS4.stWM_Power.Status := G_AXIS4.fbWM_Power.Status;

// NETWORK 5
G_AXIS4.fbWM_MoveVelocity(
    Axis := G_AXIS4.WMAxis,
    Execute := G_AXIS4.stWM_VelCmd.bExe,
    Velocity := G_AXIS4.stWM_VelCmd.lrVelocity,
    Acceleration := G_AXIS4.stWM_VelCmd.lrAcceleration,
    Deceleration := G_AXIS4.stWM_VelCmd.lrDeceleration,
    Jerk := G_AXIS4.stWM_VelCmd.lrJerk,
    Direction := G_AXIS4.stWM_VelCmd.EnuDirection,
    BufferMode := G_AXIS4.stWM_VelCmd.EnuBufferMode,
    Options := G_AXIS4.stWM_VelCmd.EnuOptions,
    Busy => G_AXIS4.stWM_MoveVelocity.Busy,
    Active => G_AXIS4.stWM_MoveVelocity.Active,
    CommandAborted => G_AXIS4.stWM_MoveVelocity.CmdAborted,
    Error => G_AXIS4.stWM_MoveVelocity.Error,
    ErrorID => G_AXIS4.stWM_MoveVelocity.ErrorID); // MC_MoveVelocity
G_AXIS4.stWM_MoveVelocity.InVelocity := G_AXIS4.fbWM_MoveVelocity.InVelocity;

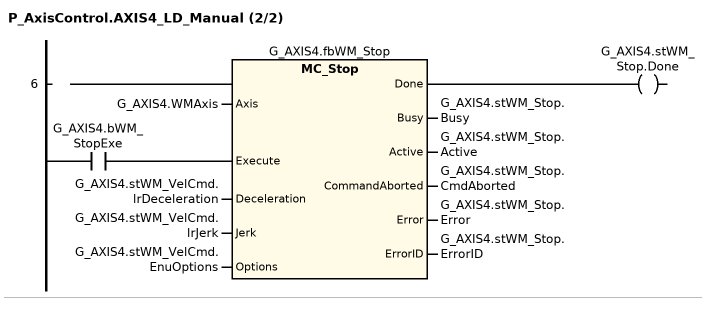
// NETWORK 6
G_AXIS4.fbWM_Stop(
    Axis := G_AXIS4.WMAxis,
    Execute := G_AXIS4.bWM_StopExe,
    Deceleration := G_AXIS4.stWM_VelCmd.lrDeceleration,
    Jerk := G_AXIS4.stWM_VelCmd.lrJerk,
    Options := G_AXIS4.stWM_VelCmd.EnuOptions,
    Busy => G_AXIS4.stWM_Stop.Busy,
    Active => G_AXIS4.stWM_Stop.Active,
    CommandAborted => G_AXIS4.stWM_Stop.CmdAborted,
    Error => G_AXIS4.stWM_Stop.Error,
    ErrorID => G_AXIS4.stWM_Stop.ErrorID); // MC_Stop
G_AXIS4.stWM_Stop.Done := G_AXIS4.fbWM_Stop.Done;
END_METHOD

METHOD Manual_mode : BOOL
VAR_INPUT
END_VAR
//Axis 1 Main arm actuator
AXIS1_LD_Manual();

G_AXIS1.bBC_ResetExe := FALSE;

G_AXIS1.stBC_VelCmd.EnuDirection := MC_Undefined_Direction;

G_AXIS1.stBC_VelCmd.bExe := FALSE;

G_AXIS1.bBC_PowerEnCmd := G_Inputs.bManualModeSelector;

IF G_Sensors.fJoystickLeftNormalizedX  > 0 AND G_Inputs.bJoystickLeftEnable THEN
	G_AXIS1.bBC_PowerEnNegative := TRUE;
	G_AXIS1.stBC_VelCmd.EnuDirection := MC_Negative_Direction;
	G_AXIS1.lrBC_PowerOverride := ABS(G_Sensors.fJoystickLeftNormalizedX) * 100;	
	G_AXIS1.stBC_VelCmd.bExe := TRUE;
ELSIF G_Sensors.fJoystickLeftNormalizedX < 0 AND G_Inputs.bJoystickLeftEnable THEN
	G_AXIS1.bBC_PowerEnPositive := TRUE;
	G_AXIS1.stBC_VelCmd.EnuDirection := MC_Positive_Direction;
	G_AXIS1.lrBC_PowerOverride := ABS(G_Sensors.fJoystickLeftNormalizedX) * 100;	
	G_AXIS1.stBC_VelCmd.bExe := TRUE;
ELSE
	 G_AXIS1.lrBC_PowerOverride := 0;
	 G_AXIS1.stBC_VelCmd.bExe := FALSE;
	 G_AXIS1.bBC_PowerEnNegative := FALSE;
	 G_AXIS1.bBC_PowerEnPositive := FALSE;
END_IF

G_AXIS1.bBC_ResetExe := TRUE;


//Axis 2 Slew joint actuator
AXIS2_LD_Manual();

G_AXIS2.bSJ_ResetExe := FALSE;

G_AXIS2.stSJ_VelCmd.EnuDirection := MC_Undefined_Direction;

G_AXIS2.stSJ_VelCmd.bExe := FALSE;

G_AXIS2.bSJ_PowerEnCmd := G_Inputs.bManualModeSelector;

IF G_Sensors.fJoystickRightNormalizedX  > 0 AND G_Inputs.bJoystickRightEnable THEN
	G_AXIS2.bSJ_PowerEnPositive := TRUE;
	G_AXIS2.stSJ_VelCmd.EnuDirection := MC_Positive_Direction;
	G_AXIS2.lrSJ_PowerOverride := ABS(G_Sensors.fJoystickRightNormalizedX) * 100;	
	G_AXIS2.stSJ_VelCmd.bExe := TRUE;
ELSIF G_Sensors.fJoystickRightNormalizedX < 0 AND G_Inputs.bJoystickRightEnable THEN
	G_AXIS2.bSJ_PowerEnNegative := TRUE;
	G_AXIS2.stSJ_VelCmd.EnuDirection := MC_Negative_Direction;
	G_AXIS2.lrSJ_PowerOverride := ABS(G_Sensors.fJoystickRightNormalizedX) * 100;	
	G_AXIS2.stSJ_VelCmd.bExe := TRUE;
ELSE
	 G_AXIS2.lrSJ_PowerOverride := 0;
	 G_AXIS2.stSJ_VelCmd.bExe := FALSE;
	 G_AXIS2.bSJ_PowerEnNegative := FALSE;
	 G_AXIS2.bSJ_PowerEnPositive := FALSE;
END_IF

G_AXIS2.bSJ_ResetExe := TRUE;


//Axis 3 Knuckle arm actuator
AXIS3_LD_Manual();

G_AXIS3.bTC_ResetExe := FALSE;

G_AXIS3.stTC_VelCmd.EnuDirection := MC_Undefined_Direction;

G_AXIS3.stTC_VelCmd.bExe := FALSE;

G_AXIS3.bTC_PowerEnCmd := G_Inputs.bManualModeSelector;

IF G_Sensors.fJoystickLeftNormalizedY  > 0 AND G_Inputs.bJoystickLeftEnable THEN
	G_AXIS3.bTC_PowerEnPositive := TRUE;
	G_AXIS3.stTC_VelCmd.EnuDirection := MC_Positive_Direction;
	G_AXIS3.lrTC_PowerOverride := ABS(G_Sensors.fJoystickLeftNormalizedY) * 100;	
	G_AXIS3.stTC_VelCmd.bExe := TRUE;
ELSIF G_Sensors.fJoystickLeftNormalizedY < 0 AND G_Inputs.bJoystickLeftEnable THEN
	G_AXIS3.bTC_PowerEnNegative := TRUE;
	G_AXIS3.stTC_VelCmd.EnuDirection := MC_Negative_Direction;
	G_AXIS3.lrTC_PowerOverride := ABS(G_Sensors.fJoystickLeftNormalizedY) * 100;	
	G_AXIS3.stTC_VelCmd.bExe := TRUE;
ELSE
	 G_AXIS3.lrTC_PowerOverride := 0;
	 G_AXIS3.stTC_VelCmd.bExe := FALSE;
	 G_AXIS3.bTC_PowerEnNegative := FALSE;
	 G_AXIS3.bTC_PowerEnPositive := FALSE;
END_IF

G_AXIS3.bTC_ResetExe := TRUE;

(*
AXIS3_LD();

GVL_AXIS3.bTC_ResetExe := G_Inputs.bJoystickLeftEnable;

GVL_AXIS3.EnuMoveVelDirection := G_Sensors.MCDirectionAxis3;

GVL_AXIS3.bTC_PowerEnCmd := G_Inputs.bManualModeSelector;
GVL_AXIS3.bTC_PowerEnNegative := G_Inputs.bManualModeSelector;
GVL_AXIS3.bTC_PowerEnPositive := G_Inputs.bManualModeSelector;


// Velocity control
IF G_Sensors.fJoystickLeftNormalizedY  > 0.01 AND G_Inputs.bJoystickLeftEnable THEN
	GVL_AXIS3.stTC_VelCmd.EnuDirection := MC_Positive_Direction;
	GVL_AXIS3.lrTC_PowerOverride := ABS(G_Sensors.fJoystickLeftNormalizedY) * 100;	
	GVL_AXIS3.stTC_VelCmd.bExe := TRUE;
ELSIF G_Sensors.fJoystickLeftNormalizedY < 0.01 AND G_Inputs.bJoystickLeftEnable THEN
	GVL_AXIS3.stTC_VelCmd.EnuDirection := MC_Negative_Direction;
	GVL_AXIS3.lrTC_PowerOverride := ABS(G_Sensors.fJoystickLeftNormalizedY) * 100;	
	GVL_AXIS3.stTC_VelCmd.bExe := TRUE;
ELSE
	 GVL_AXIS3.lrTC_PowerOverride := 0;
	 //GVL_AXIS3.stTC_VelCmd.EnuDirection := MC_Current_Direction;
	 GVL_AXIS3.stTC_VelCmd.bExe := FALSE;
END_IF
*)

(*
AXIS4_LD();

GVL_AXIS4.bWM_ResetExe := G_Inputs.bJoystickRightEnable;

GVL_AXIS4.EnuMoveVelDirection := G_Sensors.MCDirectionAxis4;

GVL_AXIS4.bWM_PowerEnCmd := G_Inputs.bManualModeSelector;
GVL_AXIS4.bWM_PowerEnNegative := G_Inputs.bManualModeSelector;
GVL_AXIS4.bWM_PowerEnPositive := G_Inputs.bManualModeSelector;


// Velocity control
IF G_Sensors.fJoystickLeftNormalizedY  > 0 AND G_Inputs.bJoystickRightEnable THEN
	GVL_AXIS4.lrWM_PowerOverride := ABS(G_Sensors.fJoystickRightNormalizedY) * 100;
	GVL_AXIS4.stWM_VelCmd.EnuDirection := MC_Positive_Direction;
	GVL_AXIS4.stWM_VelCmd.bExe := TRUE;
ELSIF G_Sensors.fJoystickLeftNormalizedY < 0 AND G_Inputs.bJoystickLeftEnable THEN
	GVL_AXIS4.lrWM_PowerOverride := ABS(G_Sensors.fJoystickLeftNormalizedY) * 100;
	GVL_AXIS4.stWM_VelCmd.EnuDirection := MC_Negative_Direction;
	GVL_AXIS4.stWM_VelCmd.bExe := TRUE;
ELSE
	 GVL_AXIS4.lrWM_PowerOverride := 0;
	 GVL_AXIS4.stWM_VelCmd.EnuDirection := MC_Current_Direction;
	 GVL_AXIS4.stWM_VelCmd.bExe := FALSE;
END_IF
*)

//Axis 4 Winch motor actuator
AXIS4_LD_Manual();

G_AXIS4.bWM_ResetExe := FALSE;

G_AXIS4.stWM_VelCmd.EnuDirection := MC_Undefined_Direction;

G_AXIS4.stWM_VelCmd.bExe := FALSE;

G_AXIS4.bWM_PowerEnCmd := G_Inputs.bManualModeSelector;

IF G_Sensors.fJoystickRightNormalizedY  > 0 AND G_Inputs.bJoystickRightEnable THEN
	G_AXIS4.bWM_PowerEnNegative := TRUE;
	G_AXIS4.stWM_VelCmd.EnuDirection := MC_Negative_Direction;
	G_AXIS4.lrWM_PowerOverride := ABS(G_Sensors.fJoystickRightNormalizedY) * 100;	
	G_AXIS4.stWM_VelCmd.bExe := TRUE;
ELSIF G_Sensors.fJoystickRightNormalizedY < 0 AND G_Inputs.bJoystickRightEnable THEN
	G_AXIS4.bWM_PowerEnPositive := TRUE;
	G_AXIS4.stWM_VelCmd.EnuDirection := MC_Positive_Direction;
	G_AXIS4.lrWM_PowerOverride := ABS(G_Sensors.fJoystickRightNormalizedY) * 100;	
	G_AXIS4.stWM_VelCmd.bExe := TRUE;
ELSE
	 G_AXIS4.lrWM_PowerOverride := 0;
	 G_AXIS4.stWM_VelCmd.bExe := FALSE;
	 G_AXIS4.bWM_PowerEnNegative := FALSE;
	 G_AXIS4.bWM_PowerEnPositive := FALSE;
END_IF

G_AXIS4.bWM_ResetExe := TRUE;
END_METHOD

METHOD Stop_mode : BOOL
VAR_INPUT
END_VAR
//Stop mode

	G_AXIS1.lrBC_PowerOverride := 0;
	G_AXIS1.bBC_StopExe := TRUE;
	G_AXIS1.bBC_PowerEnCmd := FALSE;
	
	AXIS1_LD_Auto();
	AXIS1_LD_Manual();
	
	G_AXIS2.lrSJ_PowerOverride := 0;	
	G_AXIS2.bSJ_StopExe := TRUE;	
	G_AXIS2.bSJ_PowerEnCmd := FALSE;
	
	//AXIS2_LD_Auto();
	AXIS2_LD_Manual();
	
	G_AXIS3.lrTC_PowerOverride := 0;	
	G_AXIS3.bTC_StopExe := TRUE;
	G_AXIS3.bTC_PowerEnCmd := FALSE;
	
	AXIS3_LD_Auto();
	AXIS3_LD_Manual();
	
	G_AXIS4.lrWM_PowerOverride := 0;
	G_AXIS4.bWM_StopExe := TRUE;
	G_AXIS4.bWM_PowerEnCmd := FALSE;
	
	AXIS4_LD_Auto();
	AXIS4_LD_Manual();
END_METHOD

END_PROGRAM

(* stored: Version 1.1.0.1, ProductVersion 3.1.4024.12
   POU P_AxisControl: Id {5037aaa5-6389-4d48-9944-f1b3147b0b82}, SpecialFunc None
   Method Auto_mode: Id {d04e60f4-7a42-4fb1-907e-93e16dbafa43}
   Method AXIS1_LD_Auto: Id {30907942-6a1d-4345-9aab-8829bd87d527}
   Method AXIS1_LD_Manual: Id {a2ea73c2-d9a7-46bb-9d54-a37d5bff0a65}
   Method AXIS2_LD_Manual: Id {bdec519a-41ff-484d-9600-76653e24e62b}
   Method AXIS3_LD_Auto: Id {0b7586c2-7587-4f9c-ad47-7bf16864663e}
   Method AXIS3_LD_Manual: Id {3773e93e-9c66-4353-b78a-0a74486d73ef}
   Method AXIS4_LD_Auto: Id {8b81b91c-b043-4745-82a0-5697b09e72c1}
   Method AXIS4_LD_Manual: Id {c68d9161-8577-4188-91d1-8d05a7c19713}
   Method Manual_mode: Id {1fd68a25-3da3-4bba-af59-1b4dc6fc6de5}
   Method Stop_mode: Id {3259567f-99d7-4bb9-8bb0-5bdc3da29b5d} *)
